Fanuc KAREL source: kt00080.compact.KL

PROGRAM KT00080
%STACKSIZE=65535
%PRIORITY=65535
%NOLOCKGROUP
VAR
R1 : REAL
H2 : ARRAY[2] OF SHORT
OUT : REAL
BEGIN
R1=2.0
H2[1]=3
OUT=(R1 * (H2[1]))
END KT00080
